{attribute addProperty BoxType "EL2202-0000-0016"}
{attribute addProperty Id "OutputAT %Q*BOOL811TriStateAT %Q*BOOL812"}
{attribute addProperty CRC "3560699434"}
{attribute addProperty SizeInBites "16"}
{attribute addProperty SizeInBytes "2"}
TYPE Channel_D43BF62A :
STRUCT
	{attribute addProperty Name "Output"}
	Output AT %Q* : BOOL;
	{attribute addProperty Name "TriState"}
	TriState AT %Q* : BOOL;
END_STRUCT
END_TYPE

(* stored: Version 1.2.0.0, ProductVersion 3.1.4024.9
   DUT Channel_D43BF62A: Id {65e8682d-930b-4599-8c7f-82e6d15a4849} *)
